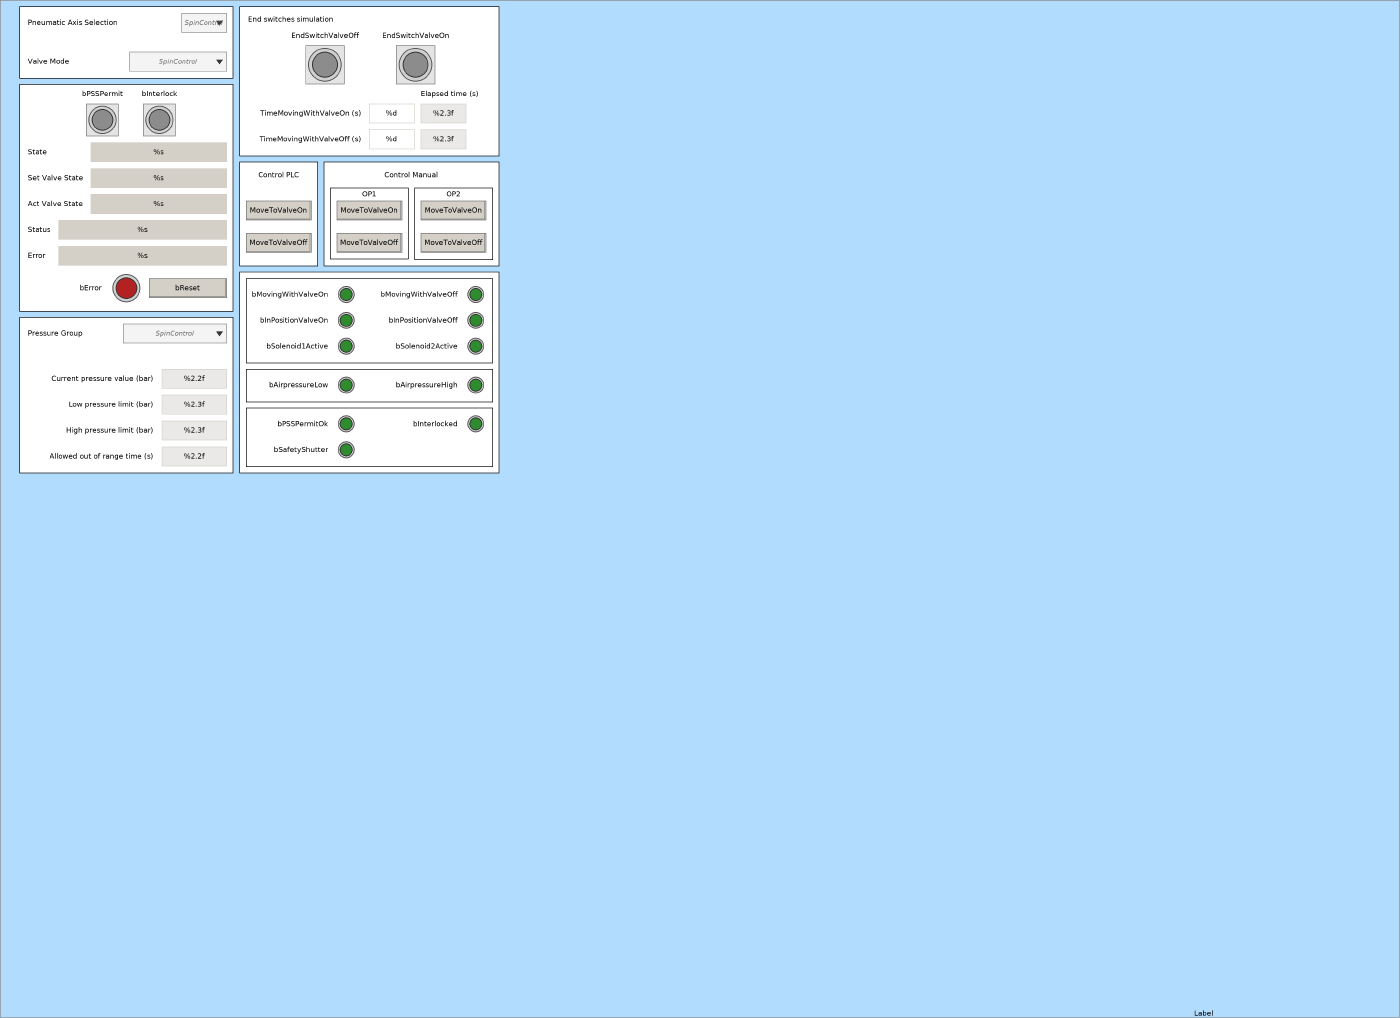
VISUALIZATION PneumaticsVisu  // 2163x1573
    Rectangle (370,420 401x311)
    Rectangle (380,430 381x131)
    Rectangle (370,250 121x161)
    Rectangle (380,630 381x91)
    Rectangle (380,570 381x51)
    Rectangle (30,10 330x111)
    Label (40,20 150x30), "Pneumatic Axis Selection"
    Rectangle (370,10 401x231)
    Label (380,20 140x20), "End switches simulation"
    SpinControl (280,20 70x30), variable: MAIN.hmiPneumaticAxisSelection
        p651134158: GVL_APP.nPNEUMATIC_AXIS_NUM
    Textfield (570,160 70x30), "%d", text variable: GVL.astPneumaticAxes[MAIN.hmiPneumaticAxisSelection].stPneumaticAxisConfig.nTimeLimitMovingWithValveOn
        OnMouseClick: write the text variable via Default
    Label (380,160 181x30), "TimeMovingWithValveOn (s)"
    Label (380,200 181x30), "TimeMovingWithValveOff (s)"
    Label (40,80 80x30), "Valve Mode"
    Rectangle (30,130 330x351)
    Label (110,430 50x30), "bError"
    Lamp1 (170,420 50x50), variable: GVL.astPneumaticAxes[MAIN.hmiPneumaticAxisSelection].stPneumaticAxisStatus.bError, style: Lamp-Lamp1-Red
    Label (40,380 31x30), "Error"
    Textfield (90,380 260x30), "%s", text variable: GVL.astPneumaticAxes[MAIN.hmiPneumaticAxisSelection].ePneumaticAxisErrors, text list: 'languageSupport'
    Label (380,250 101x41), "Control PLC"
    Label (380,440 130x30), "bMovingWithValveOn"
    Lamp1 (520,440 30x30), variable: GVL.astPneumaticAxes[MAIN.hmiPneumaticAxisSelection].stPneumaticAxisStatus.bMovingWithValveOn, style: Lamp-Lamp1-Green
    Label (580,440 130x30), "bMovingWithValveOff"
    Lamp1 (520,480 30x30), variable: GVL.astPneumaticAxes[MAIN.hmiPneumaticAxisSelection].stPneumaticAxisStatus.bInPositionValveOn, style: Lamp-Lamp1-Green
    Lamp1 (520,520 30x30), variable: GVL.astPneumaticAxes[MAIN.hmiPneumaticAxisSelection].stPneumaticAxisStatus.bSolenoid1Active, style: Lamp-Lamp1-Green
    Label (380,520 130x30), "bSolenoid1Active"
    Button (230,430 120x30), "bReset"
        OnMouseDown: execute { GVL.astPneumaticAxes[Main.hmiPneumaticAxisSelection].stPneumaticAxisControl.bReset := TRUE; }
    Label (40,220 41x30), "State"
    Textfield (140,220 210x30), "%s", text variable: MAIN.afbPneumaticAxes[MAIN.hmiPneumaticAxisSelection].eState, text list: 'languageSupport'
    Textfield (90,340 260x30), "%s", text variable: GVL.astPneumaticAxes[MAIN.hmiPneumaticAxisSelection].stPneumaticAxisStatus.sStatus, text list: 'languageSupport'
    Label (40,340 50x30), "Status"
    Textfield (570,200 70x30), "%d", text variable: GVL.astPneumaticAxes[MAIN.hmiPneumaticAxisSelection].stPneumaticAxisConfig.nTimeLimitMovingWithValveOff
        OnMouseClick: write the text variable via Default
    Textfield (650,160 70x30), "%2.3f", text variable: GVL.astPneumaticAxes[MAIN.hmiPneumaticAxisSelection].stPneumaticAxisStatus.fTimeElapsedMovingWithValveOn
    Textfield (650,200 70x30), "%2.3f", text variable: GVL.astPneumaticAxes[MAIN.hmiPneumaticAxisSelection].stPneumaticAxisStatus.fTimeElapsedMovingWithValveOff
    SpinControl (200,80 150x30), variable: GVL.astPneumaticAxes[MAIN.hmiPneumaticAxisSelection].stPneumaticAxisConfig.ePneumaticAxisMode
        p576042468: E_PneumaticAxisMode.eMonostable
        p651134158: E_PneumaticAxisMode.eBistable
    Label (640,130 110x30), "Elapsed time (s)"
    Label (450,40 105x30), "EndSwitchValveOff"
    PushSwitchLed (472,70 60x60), variable: GVL.astPneumaticAxes[MAIN.hmiPneumaticAxisSelection].stPneumaticAxisInputs.bEndSwitchValveOff, behaviour: TOGGLE, style: Switch-PushSwitchLed-Gray
    Label (590,40 105x30), "EndSwitchValveOn"
    PushSwitchLed (612,70 60x60), variable: GVL.astPneumaticAxes[MAIN.hmiPneumaticAxisSelection].stPneumaticAxisInputs.bEndSwitchValveOn, behaviour: TOGGLE, style: Switch-PushSwitchLed-Gray
    Label (123,130 71x30), "bPSSPermit"
    PushSwitchLed (133,160 50x50), variable: GVL.astPneumaticAxes[MAIN.hmiPneumaticAxisSelection].stPneumaticAxisInputs.bPSSPermitOK, behaviour: TOGGLE, style: Switch-PushSwitchLed-Gray
    PushSwitchLed (221,160 50x50), variable: GVL.astPneumaticAxes[MAIN.hmiPneumaticAxisSelection].stPneumaticAxisControl.bInterlockLatched, behaviour: TOGGLE, style: Switch-PushSwitchLed-Gray
    Label (216,130 61x30), "bInterlock"
    Label (1557,1559 606x14), "Label"
    Rectangle (500,250 271x161)
    Label (510,250 251x41), "Control Manual"
    Rectangle (640,290 121x111)
    Rectangle (510,290 121x110)
    Label (650,290 101x20), "OP2"
    Label (520,290 101x20), "OP1"
    Textfield (140,260 210x30), "%s", text variable: MAIN.afbPneumaticAxes[MAIN.hmiPneumaticAxisSelection].eSetValveState, text list: 'languageSupport'
    Label (40,260 91x30), "Set Valve State"
    Button (380,310 101x30), "MoveToValveOn"
        OnMouseDown: execute { GVL.astPneumaticAxes[Main.hmiPneumaticAxisSelection].stPneumaticAxisControl.bValveOn := TRUE; }
        OnMouseUp: execute { GVL.astPneumaticAxes[Main.hmiPneumaticAxisSelection].stPneumaticAxisControl.bValveOn := FALSE; }
    Button (380,360 101x30), "MoveToValveOff"
        OnMouseDown: execute { GVL.astPneumaticAxes[Main.hmiPneumaticAxisSelection].stPneumaticAxisControl.bValveOff := TRUE; }
        OnMouseUp: execute { GVL.astPneumaticAxes[Main.hmiPneumaticAxisSelection].stPneumaticAxisControl.bValveOff := FALSE; }
    Button (520,310 101x30), "MoveToValveOn"
        OnMouseDown: execute { GVL.astPneumaticAxes[Main.hmiPneumaticAxisSelection].stPneumaticAxisInputs.bValveOnManualOP1 := TRUE; }
        OnMouseUp: execute { GVL.astPneumaticAxes[Main.hmiPneumaticAxisSelection].stPneumaticAxisInputs.bValveOnManualOP1 := FALSE; }
    Button (520,360 101x30), "MoveToValveOff"
        OnMouseDown: execute { GVL.astPneumaticAxes[Main.hmiPneumaticAxisSelection].stPneumaticAxisInputs.bValveOffManualOP1 := TRUE; }
        OnMouseUp: execute { GVL.astPneumaticAxes[Main.hmiPneumaticAxisSelection].stPneumaticAxisInputs.bValveOffManualOP1 := FALSE; }
    Button (650,310 101x30), "MoveToValveOn"
        OnMouseDown: execute { GVL.astPneumaticAxes[Main.hmiPneumaticAxisSelection].stPneumaticAxisInputs.bValveOnManualOP2 := TRUE; }
        OnMouseUp: execute { GVL.astPneumaticAxes[Main.hmiPneumaticAxisSelection].stPneumaticAxisInputs.bValveOnManualOP2 := FALSE; }
    Button (650,360 101x30), "MoveToValveOff"
        OnMouseDown: execute { GVL.astPneumaticAxes[Main.hmiPneumaticAxisSelection].stPneumaticAxisInputs.bValveOffManualOP2 := TRUE; }
        OnMouseUp: execute { GVL.astPneumaticAxes[Main.hmiPneumaticAxisSelection].stPneumaticAxisInputs.bValveOffManualOP2 := FALSE; }
    Lamp1 (720,440 30x30), variable: GVL.astPneumaticAxes[MAIN.hmiPneumaticAxisSelection].stPneumaticAxisStatus.bMovingWithValveOff, style: Lamp-Lamp1-Green
    Lamp1 (720,480 30x30), variable: GVL.astPneumaticAxes[MAIN.hmiPneumaticAxisSelection].stPneumaticAxisStatus.bInPositionValveOff, style: Lamp-Lamp1-Green
    Lamp1 (720,520 30x30), variable: GVL.astPneumaticAxes[MAIN.hmiPneumaticAxisSelection].stPneumaticAxisStatus.bSolenoid2Active, invisible if: GVL.astPneumaticAxes[MAIN.hmiPneumaticAxisSelection].stPneumaticAxisConfig.ePneumaticAxisMode = E_PneumaticAxisMode.eMonostable, style: Lamp-Lamp1-Green
    Label (580,480 130x30), "bInPositionValveOff"
    Label (380,480 130x30), "bInPositionValveOn"
    Label (580,520 130x30), "bSolenoid2Active", invisible if: GVL.astPneumaticAxes[MAIN.hmiPneumaticAxisSelection].stPneumaticAxisConfig.ePneumaticAxisMode = E_PneumaticAxisMode.eMonostable
    Textfield (140,300 210x30), "%s", text variable: MAIN.afbPneumaticAxes[MAIN.hmiPneumaticAxisSelection].eActValveState, text list: 'languageSupport'
    Label (40,300 91x30), "Act Valve State"
    Rectangle (30,490 330x241)
    Label (50,570 190x30), "Current pressure value (bar)"
    Label (50,610 190x30), "Low pressure limit (bar)"
    Label (50,650 190x30), "High pressure limit (bar)"
    Label (30,690 210x30), "Allowed out of range time (s)"
    Textfield (250,570 100x30), "%2.2f", text variable: GVL.afbPressureGroup[GVL.astPneumaticAxes[MAIN.hmiPneumaticAxisSelection].stPneumaticAxisConfig.eSelectPneumaticAxisGroup]._fScaledPressureValue
    Textfield (250,610 100x30), "%2.3f", text variable: GVL.afbPressureGroup[GVL.astPneumaticAxes[MAIN.hmiPneumaticAxisSelection].stPneumaticAxisConfig.eSelectPneumaticAxisGroup].fPressureLimitLow
    Textfield (250,650 100x30), "%2.3f", text variable: GVL.afbPressureGroup[GVL.astPneumaticAxes[MAIN.hmiPneumaticAxisSelection].stPneumaticAxisConfig.eSelectPneumaticAxisGroup].fPressureLimitHigh
    Textfield (250,690 100x30), "%2.2f", text variable: TIME_TO_LREAL(GVL.afbPressureGroup[GVL.astPneumaticAxes[MAIN.hmiPneumaticAxisSelection].stPneumaticAxisConfig.eSelectPneumaticAxisGroup].tPressureOutOfRange)/1000.0
    Lamp1 (520,580 30x30), variable: GVL.astPneumaticAxes[MAIN.hmiPneumaticAxisSelection].stPneumaticAxisStatus.bAirPressureLow, style: Lamp-Lamp1-Green
    Label (380,580 130x30), "bAirpressureLow"
    Lamp1 (720,580 30x30), variable: GVL.astPneumaticAxes[MAIN.hmiPneumaticAxisSelection].stPneumaticAxisStatus.bAirPressureHigh, style: Lamp-Lamp1-Green
    Label (580,580 130x30), "bAirpressureHigh"
    Lamp1 (520,640 30x30), variable: GVL.astPneumaticAxes[MAIN.hmiPneumaticAxisSelection].stPneumaticAxisStatus.bPSSPermitOK, style: Lamp-Lamp1-Green
    Label (380,640 130x30), "bPSSPermitOk"
    Lamp1 (720,640 30x30), variable: GVL.astPneumaticAxes[MAIN.hmiPneumaticAxisSelection].stPneumaticAxisStatus.bInterlocked, style: Lamp-Lamp1-Green
    Label (580,640 130x30), "bInterlocked"
    Lamp1 (520,680 30x30), variable: GVL.astPneumaticAxes[MAIN.hmiPneumaticAxisSelection].stPneumaticAxisConfig.bSafetyShutter, style: Lamp-Lamp1-Green
    Label (380,680 130x30), "bSafetyShutter"
    Label (40,500 230x30), "Pressure Group"
    SpinControl (190,500 160x30), variable: GVL.astPneumaticAxes[MAIN.hmiPneumaticAxisSelection].stPneumaticAxisConfig.eSelectPneumaticAxisGroup
        p576042468: E_PneumaticAxisGroup.ePneumaticAxisGroup1
        p651134158: E_PneumaticAxisGroup.ePneumaticAxisGroup2
END_VISUALIZATION

(* stored: Version 1.1.0.1
   Visu PneumaticsVisu: Id {957f9dde-5850-0da0-173d-164c7d8c0b2d} *)
